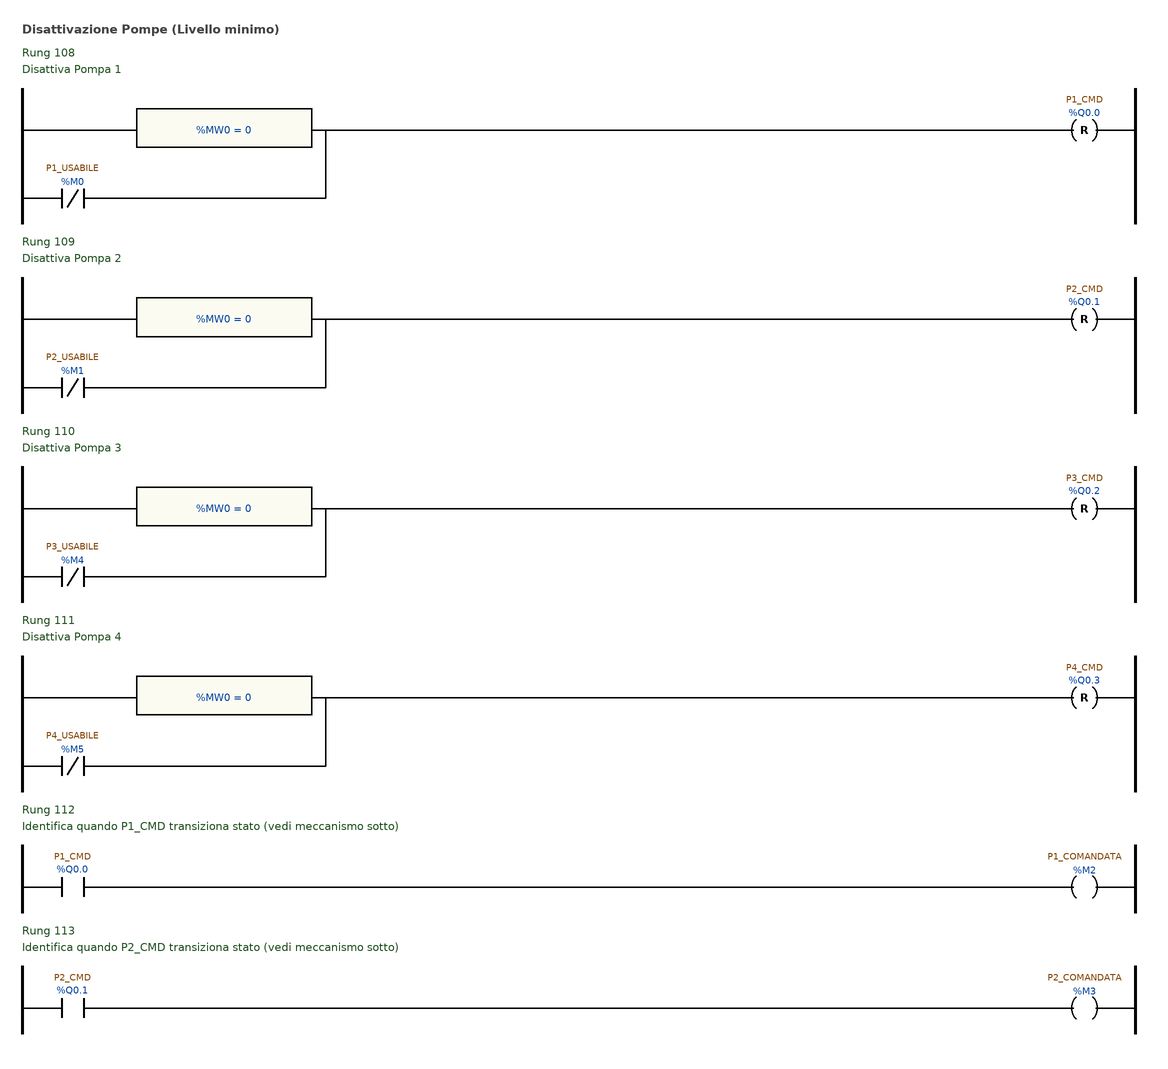
[picture p24: Disattivazione Pompe (Livello minimo), ladder]

// Rung 108
// Disattiva Pompa 1
  LD [ %MW0 = 0 ]         (* NUM_POMPE_DA_COMANDARE *)
  ORN %M0                 (* P1_USABILE *)
  R %Q0.0                 (* P1_CMD *)
  // as ST:
  //   IF NUM_POMPE_DA_COMANDARE = 0 OR NOT P1_USABILE THEN P1_CMD := FALSE; END_IF;

// Rung 109
// Disattiva Pompa 2
  LD [ %MW0 = 0 ]         (* NUM_POMPE_DA_COMANDARE *)
  ORN %M1                 (* P2_USABILE *)
  R %Q0.1                 (* P2_CMD *)
  // as ST:
  //   IF NUM_POMPE_DA_COMANDARE = 0 OR NOT P2_USABILE THEN P2_CMD := FALSE; END_IF;

// Rung 110
// Disattiva Pompa 3
  LD [ %MW0 = 0 ]         (* NUM_POMPE_DA_COMANDARE *)
  ORN %M4                 (* P3_USABILE *)
  R %Q0.2                 (* P3_CMD *)
  // as ST:
  //   IF NUM_POMPE_DA_COMANDARE = 0 OR NOT P3_USABILE THEN P3_CMD := FALSE; END_IF;

// Rung 111
// Disattiva Pompa 4
  LD [ %MW0 = 0 ]         (* NUM_POMPE_DA_COMANDARE *)
  ORN %M5                 (* P4_USABILE *)
  R %Q0.3                 (* P4_CMD *)
  // as ST:
  //   IF NUM_POMPE_DA_COMANDARE = 0 OR NOT P4_USABILE THEN P4_CMD := FALSE; END_IF;

// Rung 112
// Identifica quando P1_CMD transiziona stato (vedi meccanismo sotto)
  LD %Q0.0                (* P1_CMD *)
  ST %M2                  (* P1_COMANDATA *)
  // as ST:
  //   P1_COMANDATA := P1_CMD;

// Rung 113
// Identifica quando P2_CMD transiziona stato (vedi meccanismo sotto)
  LD %Q0.1                (* P2_CMD *)
  ST %M3                  (* P2_COMANDATA *)
  // as ST:
  //   P2_COMANDATA := P2_CMD;

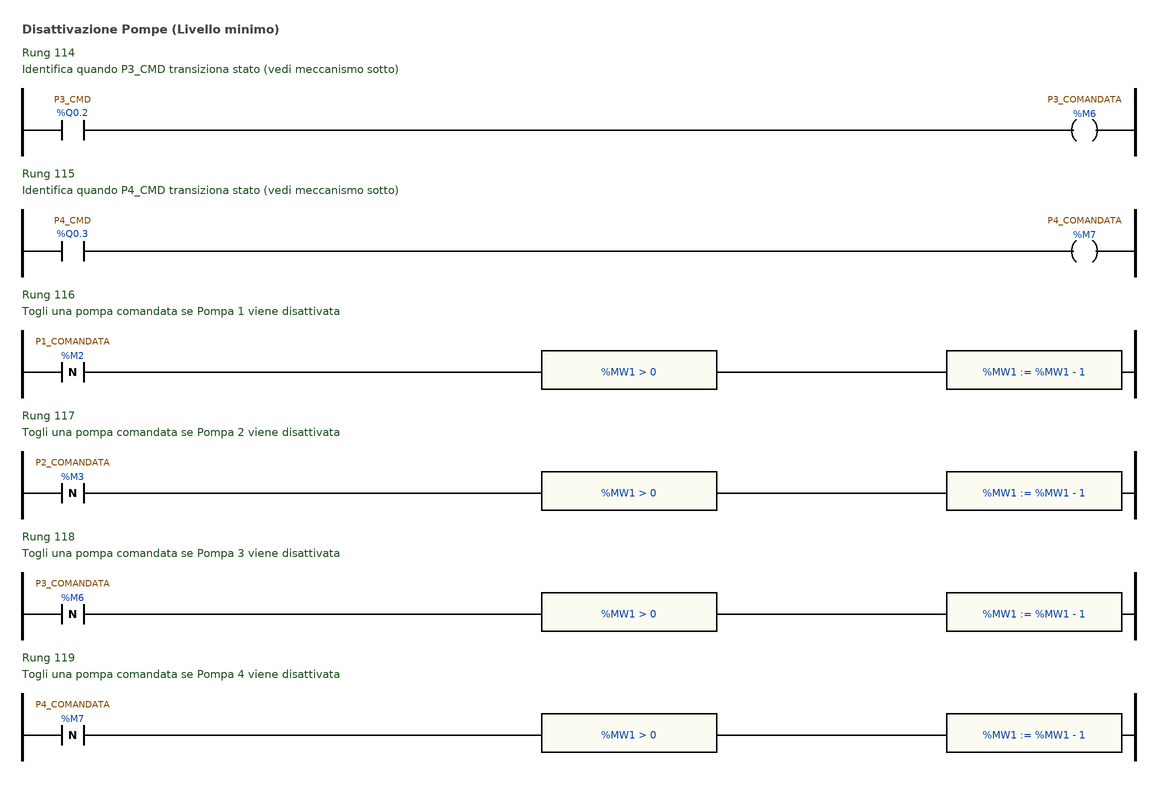

// Rung 114
// Identifica quando P3_CMD transiziona stato (vedi meccanismo sotto)
  LD %Q0.2                (* P3_CMD *)
  ST %M6                  (* P3_COMANDATA *)
  // as ST:
  //   P3_COMANDATA := P3_CMD;

// Rung 115
// Identifica quando P4_CMD transiziona stato (vedi meccanismo sotto)
  LD %Q0.3                (* P4_CMD *)
  ST %M7                  (* P4_COMANDATA *)
  // as ST:
  //   P4_COMANDATA := P4_CMD;

// Rung 116
// Togli una pompa comandata se Pompa 1 viene disattivata
  LDF %M2                 (* P1_COMANDATA *)
  AND [ %MW1 > 0 ]        (* NUM_POMPE_COMANDATE *)
  [ %MW1 := %MW1 - 1 ]    (* NUM_POMPE_COMANDATE, NUM_POMPE_COMANDATE *)
  // as ST:
  //   IF FALLING(P1_COMANDATA) AND NUM_POMPE_COMANDATE > 0 THEN NUM_POMPE_COMANDATE := NUM_POMPE_COMANDATE - 1; END_IF;

// Rung 117
// Togli una pompa comandata se Pompa 2 viene disattivata
  LDF %M3                 (* P2_COMANDATA *)
  AND [ %MW1 > 0 ]        (* NUM_POMPE_COMANDATE *)
  [ %MW1 := %MW1 - 1 ]    (* NUM_POMPE_COMANDATE, NUM_POMPE_COMANDATE *)
  // as ST:
  //   IF FALLING(P2_COMANDATA) AND NUM_POMPE_COMANDATE > 0 THEN NUM_POMPE_COMANDATE := NUM_POMPE_COMANDATE - 1; END_IF;

// Rung 118
// Togli una pompa comandata se Pompa 3 viene disattivata
  LDF %M6                 (* P3_COMANDATA *)
  AND [ %MW1 > 0 ]        (* NUM_POMPE_COMANDATE *)
  [ %MW1 := %MW1 - 1 ]    (* NUM_POMPE_COMANDATE, NUM_POMPE_COMANDATE *)
  // as ST:
  //   IF FALLING(P3_COMANDATA) AND NUM_POMPE_COMANDATE > 0 THEN NUM_POMPE_COMANDATE := NUM_POMPE_COMANDATE - 1; END_IF;

// Rung 119
// Togli una pompa comandata se Pompa 4 viene disattivata
  LDF %M7                 (* P4_COMANDATA *)
  AND [ %MW1 > 0 ]        (* NUM_POMPE_COMANDATE *)
  [ %MW1 := %MW1 - 1 ]    (* NUM_POMPE_COMANDATE, NUM_POMPE_COMANDATE *)
  // as ST:
  //   IF FALLING(P4_COMANDATA) AND NUM_POMPE_COMANDATE > 0 THEN NUM_POMPE_COMANDATE := NUM_POMPE_COMANDATE - 1; END_IF;

Subroutine Soglie (Livello minimo)
  (* SectionNumber=21, Number=19 *)

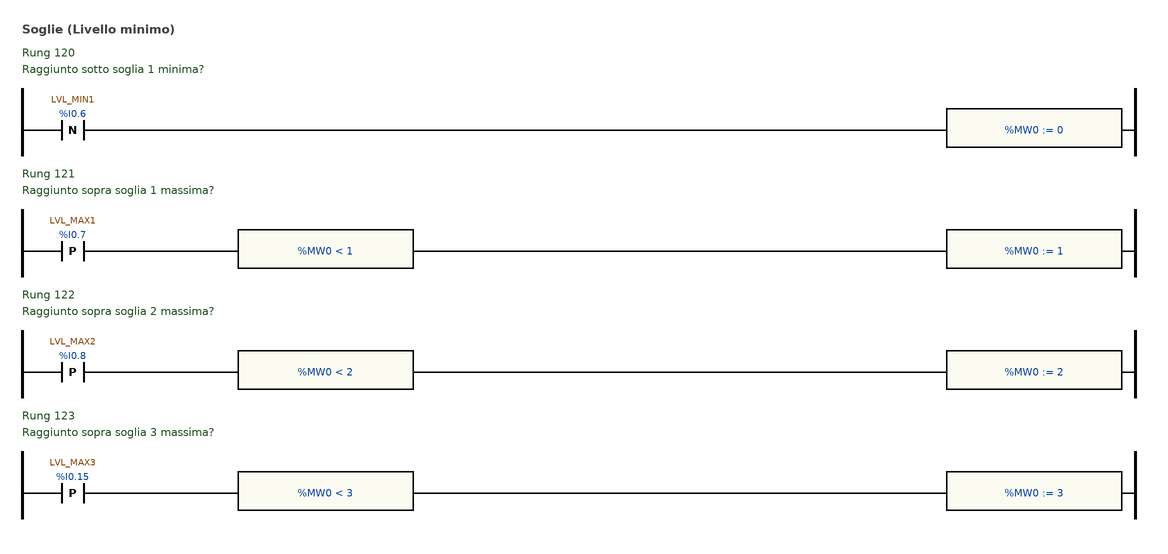

// Rung 120
// Raggiunto sotto soglia 1 minima?
  LDF %I0.6               (* LVL_MIN1 *)
  [ %MW0 := 0 ]           (* NUM_POMPE_DA_COMANDARE *)
  // as ST:
  //   IF FALLING(LVL_MIN1) THEN NUM_POMPE_DA_COMANDARE := 0; END_IF;

// Rung 121
// Raggiunto sopra soglia 1 massima?
  LDR %I0.7               (* LVL_MAX1 *)
  AND [ %MW0 < 1 ]        (* NUM_POMPE_DA_COMANDARE *)
  [ %MW0 := 1 ]           (* NUM_POMPE_DA_COMANDARE *)
  // as ST:
  //   IF RISING(LVL_MAX1) AND NUM_POMPE_DA_COMANDARE < 1 THEN NUM_POMPE_DA_COMANDARE := 1; END_IF;

// Rung 122
// Raggiunto sopra soglia 2 massima?
  LDR %I0.8               (* LVL_MAX2 *)
  AND [ %MW0 < 2 ]        (* NUM_POMPE_DA_COMANDARE *)
  [ %MW0 := 2 ]           (* NUM_POMPE_DA_COMANDARE *)
  // as ST:
  //   IF RISING(LVL_MAX2) AND NUM_POMPE_DA_COMANDARE < 2 THEN NUM_POMPE_DA_COMANDARE := 2; END_IF;

// Rung 123
// Raggiunto sopra soglia 3 massima?
  LDR %I0.15              (* LVL_MAX3 *)
  AND [ %MW0 < 3 ]        (* NUM_POMPE_DA_COMANDARE *)
  [ %MW0 := 3 ]           (* NUM_POMPE_DA_COMANDARE *)
  // as ST:
  //   IF RISING(LVL_MAX3) AND NUM_POMPE_DA_COMANDARE < 3 THEN NUM_POMPE_DA_COMANDARE := 3; END_IF;

Subroutine Ordine: Terza Pompa (Livello minimo)
  (* SectionNumber=0, Number=20 *)

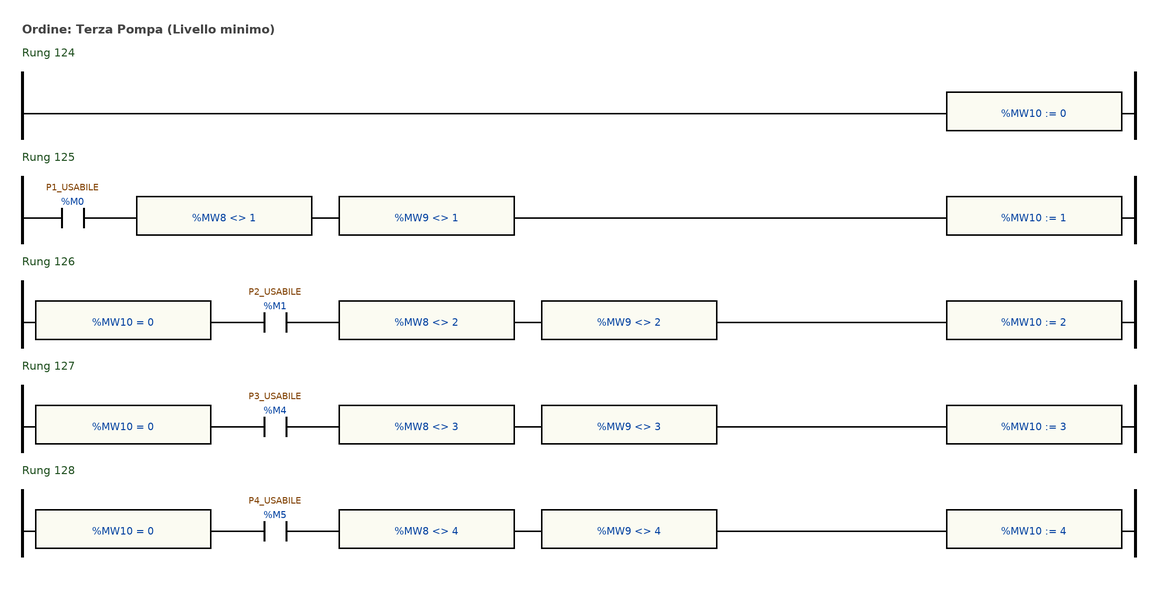

// Rung 124
  LD 1
  [ %MW10 := 0 ]          (* ORDINE_TERZA_POMPA *)
  // as ST:
  //   ORDINE_TERZA_POMPA := 0;

// Rung 125
  LD %M0                  (* P1_USABILE *)
  AND [ %MW8 <> 1 ]       (* ORDINE_PRIMA_POMPA *)
  AND [ %MW9 <> 1 ]       (* ORDINE_SECONDA_POMPA *)
  [ %MW10 := 1 ]          (* ORDINE_TERZA_POMPA *)
  // as ST:
  //   IF P1_USABILE AND ORDINE_PRIMA_POMPA <> 1 AND ORDINE_SECONDA_POMPA <> 1 THEN ORDINE_TERZA_POMPA := 1; END_IF;

// Rung 126
  LD [ %MW10 = 0 ]        (* ORDINE_TERZA_POMPA *)
  AND %M1                 (* P2_USABILE *)
  AND [ %MW8 <> 2 ]       (* ORDINE_PRIMA_POMPA *)
  AND [ %MW9 <> 2 ]       (* ORDINE_SECONDA_POMPA *)
  [ %MW10 := 2 ]          (* ORDINE_TERZA_POMPA *)
  // as ST:
  //   IF ORDINE_TERZA_POMPA = 0 AND P2_USABILE AND ORDINE_PRIMA_POMPA <> 2 AND ORDINE_SECONDA_POMPA <> 2 THEN ORDINE_TERZA_POMPA := 2; END_IF;

// Rung 127
  LD [ %MW10 = 0 ]        (* ORDINE_TERZA_POMPA *)
  AND %M4                 (* P3_USABILE *)
  AND [ %MW8 <> 3 ]       (* ORDINE_PRIMA_POMPA *)
  AND [ %MW9 <> 3 ]       (* ORDINE_SECONDA_POMPA *)
  [ %MW10 := 3 ]          (* ORDINE_TERZA_POMPA *)
  // as ST:
  //   IF ORDINE_TERZA_POMPA = 0 AND P3_USABILE AND ORDINE_PRIMA_POMPA <> 3 AND ORDINE_SECONDA_POMPA <> 3 THEN ORDINE_TERZA_POMPA := 3; END_IF;

// Rung 128
  LD [ %MW10 = 0 ]        (* ORDINE_TERZA_POMPA *)
  AND %M5                 (* P4_USABILE *)
  AND [ %MW8 <> 4 ]       (* ORDINE_PRIMA_POMPA *)
  AND [ %MW9 <> 4 ]       (* ORDINE_SECONDA_POMPA *)
  [ %MW10 := 4 ]          (* ORDINE_TERZA_POMPA *)
  // as ST:
  //   IF ORDINE_TERZA_POMPA = 0 AND P4_USABILE AND ORDINE_PRIMA_POMPA <> 4 AND ORDINE_SECONDA_POMPA <> 4 THEN ORDINE_TERZA_POMPA := 4; END_IF;

Subroutine Comanda: Terza Pompa (Livello minimo)
  (* SectionNumber=0, Number=21 *)

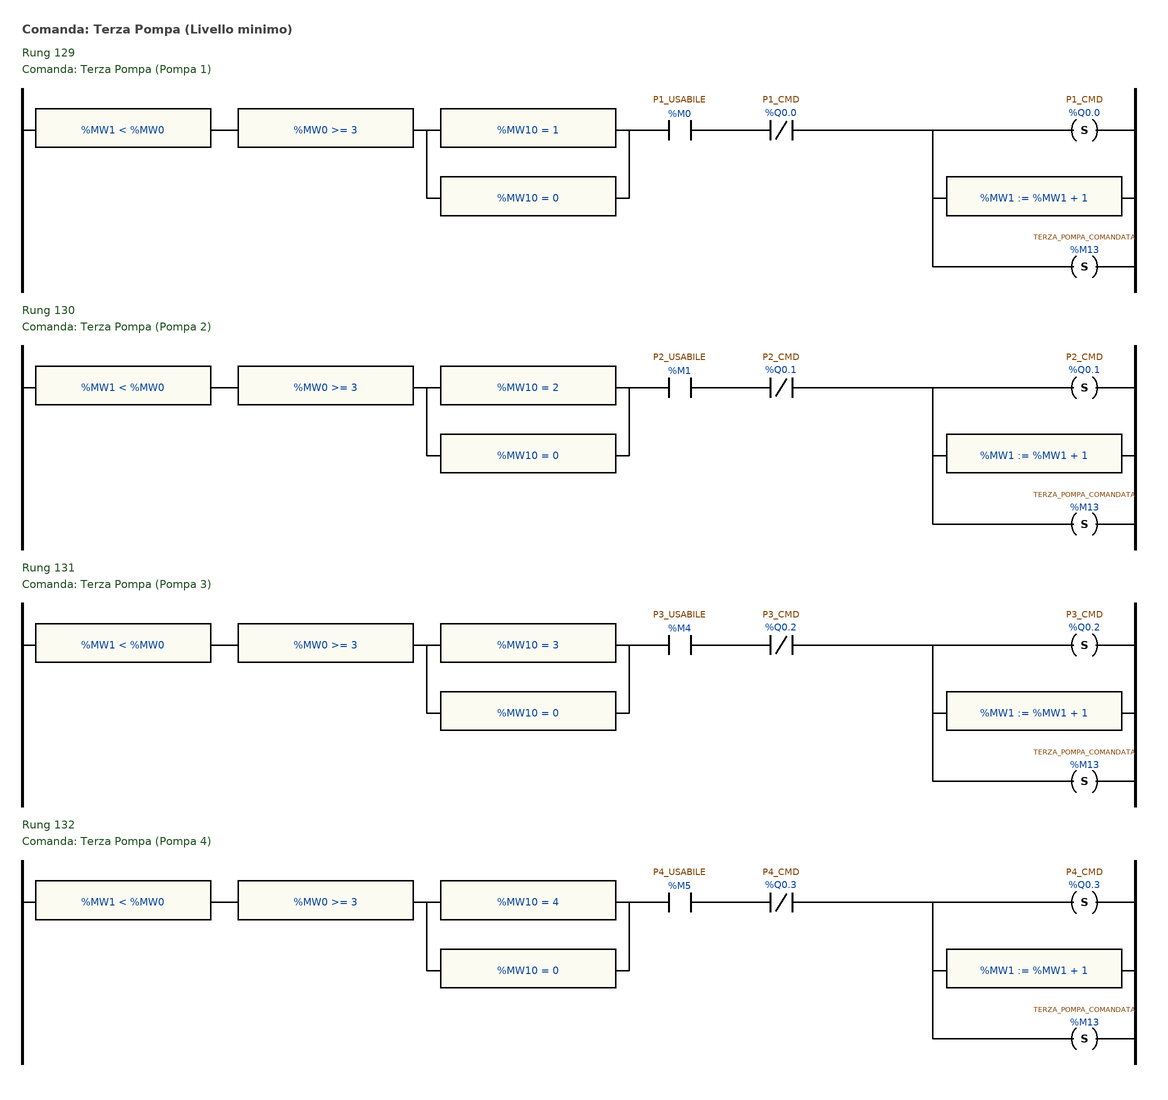

// Rung 129
// Comanda: Terza Pompa (Pompa 1)
  LD [ %MW1 < %MW0 ]      (* NUM_POMPE_COMANDATE, NUM_POMPE_DA_COMANDARE *)
  AND [ %MW0 >= 3 ]       (* NUM_POMPE_DA_COMANDARE *)
  AND( [ %MW10 = 1 ]      (* ORDINE_TERZA_POMPA *)
  OR [ %MW10 = 0 ]        (* ORDINE_TERZA_POMPA *)
  )
  AND %M0                 (* P1_USABILE *)
  ANDN %Q0.0              (* P1_CMD *)
  S %Q0.0                 (* P1_CMD *)
  [ %MW1 := %MW1 + 1 ]    (* NUM_POMPE_COMANDATE, NUM_POMPE_COMANDATE *)
  S %M13                  (* TERZA_POMPA_COMANDATA *)
  // as ST:
  //   _t1 := NUM_POMPE_COMANDATE < NUM_POMPE_DA_COMANDARE AND NUM_POMPE_DA_COMANDARE >= 3 AND (ORDINE_TERZA_POMPA = 1 OR ORDINE_TERZA_POMPA = 0) AND P1_USABILE AND NOT P1_CMD;
  //   IF _t1 THEN P1_CMD := TRUE; END_IF;
  //   IF _t1 THEN NUM_POMPE_COMANDATE := NUM_POMPE_COMANDATE + 1; END_IF;
  //   IF _t1 THEN TERZA_POMPA_COMANDATA := TRUE; END_IF;

// Rung 130
// Comanda: Terza Pompa (Pompa 2)
  LD [ %MW1 < %MW0 ]      (* NUM_POMPE_COMANDATE, NUM_POMPE_DA_COMANDARE *)
  AND [ %MW0 >= 3 ]       (* NUM_POMPE_DA_COMANDARE *)
  AND( [ %MW10 = 2 ]      (* ORDINE_TERZA_POMPA *)
  OR [ %MW10 = 0 ]        (* ORDINE_TERZA_POMPA *)
  )
  AND %M1                 (* P2_USABILE *)
  ANDN %Q0.1              (* P2_CMD *)
  S %Q0.1                 (* P2_CMD *)
  [ %MW1 := %MW1 + 1 ]    (* NUM_POMPE_COMANDATE, NUM_POMPE_COMANDATE *)
  S %M13                  (* TERZA_POMPA_COMANDATA *)
  // as ST:
  //   _t1 := NUM_POMPE_COMANDATE < NUM_POMPE_DA_COMANDARE AND NUM_POMPE_DA_COMANDARE >= 3 AND (ORDINE_TERZA_POMPA = 2 OR ORDINE_TERZA_POMPA = 0) AND P2_USABILE AND NOT P2_CMD;
  //   IF _t1 THEN P2_CMD := TRUE; END_IF;
  //   IF _t1 THEN NUM_POMPE_COMANDATE := NUM_POMPE_COMANDATE + 1; END_IF;
  //   IF _t1 THEN TERZA_POMPA_COMANDATA := TRUE; END_IF;

// Rung 131
// Comanda: Terza Pompa (Pompa 3)
  LD [ %MW1 < %MW0 ]      (* NUM_POMPE_COMANDATE, NUM_POMPE_DA_COMANDARE *)
  AND [ %MW0 >= 3 ]       (* NUM_POMPE_DA_COMANDARE *)
  AND( [ %MW10 = 3 ]      (* ORDINE_TERZA_POMPA *)
  OR [ %MW10 = 0 ]        (* ORDINE_TERZA_POMPA *)
  )
  AND %M4                 (* P3_USABILE *)
  ANDN %Q0.2              (* P3_CMD *)
  S %Q0.2                 (* P3_CMD *)
  [ %MW1 := %MW1 + 1 ]    (* NUM_POMPE_COMANDATE, NUM_POMPE_COMANDATE *)
  S %M13                  (* TERZA_POMPA_COMANDATA *)
  // as ST:
  //   _t1 := NUM_POMPE_COMANDATE < NUM_POMPE_DA_COMANDARE AND NUM_POMPE_DA_COMANDARE >= 3 AND (ORDINE_TERZA_POMPA = 3 OR ORDINE_TERZA_POMPA = 0) AND P3_USABILE AND NOT P3_CMD;
  //   IF _t1 THEN P3_CMD := TRUE; END_IF;
  //   IF _t1 THEN NUM_POMPE_COMANDATE := NUM_POMPE_COMANDATE + 1; END_IF;
  //   IF _t1 THEN TERZA_POMPA_COMANDATA := TRUE; END_IF;

// Rung 132
// Comanda: Terza Pompa (Pompa 4)
  LD [ %MW1 < %MW0 ]      (* NUM_POMPE_COMANDATE, NUM_POMPE_DA_COMANDARE *)
  AND [ %MW0 >= 3 ]       (* NUM_POMPE_DA_COMANDARE *)
  AND( [ %MW10 = 4 ]      (* ORDINE_TERZA_POMPA *)
  OR [ %MW10 = 0 ]        (* ORDINE_TERZA_POMPA *)
  )
  AND %M5                 (* P4_USABILE *)
  ANDN %Q0.3              (* P4_CMD *)
  S %Q0.3                 (* P4_CMD *)
  [ %MW1 := %MW1 + 1 ]    (* NUM_POMPE_COMANDATE, NUM_POMPE_COMANDATE *)
  S %M13                  (* TERZA_POMPA_COMANDATA *)
  // as ST:
  //   _t1 := NUM_POMPE_COMANDATE < NUM_POMPE_DA_COMANDARE AND NUM_POMPE_DA_COMANDARE >= 3 AND (ORDINE_TERZA_POMPA = 4 OR ORDINE_TERZA_POMPA = 0) AND P4_USABILE AND NOT P4_CMD;
  //   IF _t1 THEN P4_CMD := TRUE; END_IF;
  //   IF _t1 THEN NUM_POMPE_COMANDATE := NUM_POMPE_COMANDATE + 1; END_IF;
  //   IF _t1 THEN TERZA_POMPA_COMANDATA := TRUE; END_IF;
